{attribute 'qualified_only'}
VAR_GLOBAL
	senControlElement1Start		: FB_IOSensor_NO;
	senControlElement1End		: FB_IOSensor_NO;
	fbControlElement1			: FB_ControlElement1 (
									itfsenStart	:= senControlElement1Start,
	                                itfsenEnd	:= senControlElement1End
								);
	senControlElement2Start		: FB_IOSensor_NO;
	senControlElement2End		: FB_IOSensor_NO;
	senControlElement2Position1	: FB_IOSensor_NO;
	senControlElement2Position2	: FB_IOSensor_NO;
	fbControlElement2			:  FB_ControlElement2 (
									itfsenStart		:= senControlElement2Start,
	                                itfsenEnd		:= senControlElement2End,
	                                itfsenPosition1	:= senControlElement2Position1,
								    itfsenPosition2	:= senControlElement2Position2
								);

	senTopElement1Position1		: FB_IOSensor_NO;
	senTopElement1Position2		: FB_IOSensor_NO;
	fbTopElement1				: FB_TopElement1 (
									itfControlElement1		:= fbControlElement1,
								    itfControlElement2		:= fbControlElement2,
		                           	itfsenElementPosition1	:= senTopElement1Position1,
                                    itfsenElementPosition2	:= senTopElement1Position2
								);
END_VAR

(* stored: Version 1.1.0.1, ProductVersion 3.1.4024.15
   GVL GVL_TopElement1: Id {c3d2e9f1-7e99-4571-9b5c-20f4145bd99b} *)
